# EPICS autosave request: db/Rigaku_MM003i_settings.req
$(P)$(T):voltage
$(P)$(T):current
